// TwinCAT 3 PLC project Xplanar
// ProgramVersion: 3.1.4026.9
// CompilerDefines: VISU_USEPROPERTYINFO
// libraries:
//   CmpBitmapPool, * (System)
//   Tc2_Standard, * (Beckhoff Automation GmbH)
//   Tc2_System, * (Beckhoff Automation GmbH)
//   Tc2_Utilities, * (Beckhoff Automation GmbH)
//   Tc3_Mc3PlanarMotion, * (Beckhoff Automation GmbH)
//   Tc3_Physics, * (Beckhoff Automation GmbH)
//   Tc3_XPlanarUtility, * (Beckhoff Automation GmbH)
//   VisuDialogs, * (System)
//   VisuSymbols, 4.5.0.0 (System)
// project tree:
//   DUTs/ TurtleNames.TcDUT
//   / GlobalTextList.TcGTLO, ImagePool.TcIPO (not stored), PlcTask.TcTTO
//   GVLs/ GVL.TcGVL
//   POUs/ HMI_UpdateMoverStatus.TcPOU, MAIN.TcPOU, randnum.TcPOU, Traffic_Light.TcPOU, WinnersList.TcPOU, Winner_Display.TcPOU
// real-time tasks:
//   TASK XPlanar Task3: cycle T#250us, priority 1, ADS port 350
//   TASK MC-Task (MET): cycle T#2ms, priority 2, ADS port 351
//   TASK MC-Task (MPT): cycle T#10ms, priority 3, ADS port 352
//   TASK Job Task: cycle default, priority 4
//   TASK MC-Task (MET)_1: cycle T#2ms, priority 5, ADS port 521
//   TASK MC-Task (MPT)_1: cycle T#10ms, priority 10, ADS port 531
//   TASK PlcTask: cycle T#10ms, priority 20, ADS port 353
// I/O:
//   DEVICE Device 1 (EtherCAT), AmsNetId 172.18.137.9.2.1
//     Box 1 (EP2316-0003) [EP2316-0003 8 Ch. Dig. In, 10µs, 8Ch. Dig. Out 24V, 0,5A, Diagnostic, 10-Pole Plug Connector]
//   DEVICE Device 2 (EtherCAT), AmsNetId 172.18.137.9.3.1
//     Term 2 (APS4322-7000) [APS4322-7000 Drive]
//       Term 3 (APS4322-5000) [APS4322-5000 Feedback]
//     Term 4 (APS4322-7000) [APS4322-7000 Drive]
//       Term 5 (APS4322-5000) [APS4322-5000 Feedback]
// variable links:
//   Device 2 (EtherCAT) <-> TcCOM Objects/XPlanar/Part1/Tile1
//     Term 2 (APS4322-7000)/APS Comm Inputs/CommStatusWord <-> Data Pointer/MoverCommStatusWord
//     Term 2 (APS4322-7000)/APS Comm Inputs/Data {1..4} <-> Data Pointer/MoverCommDataIn[{0..3}]  (4 links)
//     Term 2 (APS4322-7000)/APS Comm Outputs/CommControlWord <-> Data Pointer/MoverCommControlWord
//     Term 2 (APS4322-7000)/APS Comm Outputs/Data 1 <-> Data Pointer/MoverCommDataOut
//     Term 2 (APS4322-7000)/APS Diagdata/DC Link Voltage <-> Data Pointer/DcLinkVoltage
//     Term 2 (APS4322-7000)/APS Diagdata/Power supply current <-> Data Pointer/PowerSupplyCurrent
//     Term 2 (APS4322-7000)/APS Inputs/StatusWord <-> Data Pointer/PowerUnitStatusWord
//     Term 2 (APS4322-7000)/APS Outputs/ControlWord <-> Data Pointer/PowerUnitControlWord
//     Term 2 (APS4322-7000)/APS Outputs/Current D 0X0 <-> Data Pointer/DCurrentSetPoints[0]
//     Term 2 (APS4322-7000)/APS Outputs/Current D 0X1 <-> Data Pointer/DCurrentSetPoints[1]
//     Term 2 (APS4322-7000)/APS Outputs/Current D 0X2 <-> Data Pointer/DCurrentSetPoints[2]
//     Term 2 (APS4322-7000)/APS Outputs/Current D 1X0 <-> Data Pointer/DCurrentSetPoints[6]
//     Term 2 (APS4322-7000)/APS Outputs/Current D 1X1 <-> Data Pointer/DCurrentSetPoints[7]
//     Term 2 (APS4322-7000)/APS Outputs/Current D 1X2 <-> Data Pointer/DCurrentSetPoints[8]
//     Term 2 (APS4322-7000)/APS Outputs/Current D 2X0 <-> Data Pointer/DCurrentSetPoints[12]
//     Term 2 (APS4322-7000)/APS Outputs/Current D 2X1 <-> Data Pointer/DCurrentSetPoints[13]
//     Term 2 (APS4322-7000)/APS Outputs/Current D 2X2 <-> Data Pointer/DCurrentSetPoints[14]
//     Term 2 (APS4322-7000)/APS Outputs/Current D 3X0 <-> Data Pointer/DCurrentSetPoints[18]
//     Term 2 (APS4322-7000)/APS Outputs/Current D 3X1 <-> Data Pointer/DCurrentSetPoints[19]
//     Term 2 (APS4322-7000)/APS Outputs/Current D 3X2 <-> Data Pointer/DCurrentSetPoints[20]
//     Term 2 (APS4322-7000)/APS Outputs/Current D 0Y0 <-> Data Pointer/DCurrentSetPoints[3]
//     Term 2 (APS4322-7000)/APS Outputs/Current D 0Y1 <-> Data Pointer/DCurrentSetPoints[4]
//     Term 2 (APS4322-7000)/APS Outputs/Current D 0Y2 <-> Data Pointer/DCurrentSetPoints[5]
//     Term 2 (APS4322-7000)/APS Outputs/Current D 1Y0 <-> Data Pointer/DCurrentSetPoints[9]
//     Term 2 (APS4322-7000)/APS Outputs/Current D 1Y1 <-> Data Pointer/DCurrentSetPoints[10]
//     Term 2 (APS4322-7000)/APS Outputs/Current D 1Y2 <-> Data Pointer/DCurrentSetPoints[11]
//     Term 2 (APS4322-7000)/APS Outputs/Current D 2Y0 <-> Data Pointer/DCurrentSetPoints[15]
//     Term 2 (APS4322-7000)/APS Outputs/Current D 2Y1 <-> Data Pointer/DCurrentSetPoints[16]
//     Term 2 (APS4322-7000)/APS Outputs/Current D 2Y2 <-> Data Pointer/DCurrentSetPoints[17]
//     Term 2 (APS4322-7000)/APS Outputs/Current D 3Y0 <-> Data Pointer/DCurrentSetPoints[21]
//     Term 2 (APS4322-7000)/APS Outputs/Current D 3Y1 <-> Data Pointer/DCurrentSetPoints[22]
//     Term 2 (APS4322-7000)/APS Outputs/Current D 3Y2 <-> Data Pointer/DCurrentSetPoints[23]
//     Term 2 (APS4322-7000)/APS Outputs/Current Q 0X0 <-> Data Pointer/QCurrentSetPoints[0]
//     Term 2 (APS4322-7000)/APS Outputs/Current Q 0X1 <-> Data Pointer/QCurrentSetPoints[1]
//     Term 2 (APS4322-7000)/APS Outputs/Current Q 0X2 <-> Data Pointer/QCurrentSetPoints[2]
//     Term 2 (APS4322-7000)/APS Outputs/Current Q 1X0 <-> Data Pointer/QCurrentSetPoints[6]
//     Term 2 (APS4322-7000)/APS Outputs/Current Q 1X1 <-> Data Pointer/QCurrentSetPoints[7]
//     Term 2 (APS4322-7000)/APS Outputs/Current Q 1X2 <-> Data Pointer/QCurrentSetPoints[8]
//     Term 2 (APS4322-7000)/APS Outputs/Current Q 2X0 <-> Data Pointer/QCurrentSetPoints[12]
//     Term 2 (APS4322-7000)/APS Outputs/Current Q 2X1 <-> Data Pointer/QCurrentSetPoints[13]
//     Term 2 (APS4322-7000)/APS Outputs/Current Q 2X2 <-> Data Pointer/QCurrentSetPoints[14]
//     Term 2 (APS4322-7000)/APS Outputs/Current Q 3X0 <-> Data Pointer/QCurrentSetPoints[18]
//     Term 2 (APS4322-7000)/APS Outputs/Current Q 3X1 <-> Data Pointer/QCurrentSetPoints[19]
//     Term 2 (APS4322-7000)/APS Outputs/Current Q 3X2 <-> Data Pointer/QCurrentSetPoints[20]
//     Term 2 (APS4322-7000)/APS Outputs/Current Q 0Y0 <-> Data Pointer/QCurrentSetPoints[3]
//     Term 2 (APS4322-7000)/APS Outputs/Current Q 0Y1 <-> Data Pointer/QCurrentSetPoints[4]
//     Term 2 (APS4322-7000)/APS Outputs/Current Q 0Y2 <-> Data Pointer/QCurrentSetPoints[5]
//     Term 2 (APS4322-7000)/APS Outputs/Current Q 1Y0 <-> Data Pointer/QCurrentSetPoints[9]
//     Term 2 (APS4322-7000)/APS Outputs/Current Q 1Y1 <-> Data Pointer/QCurrentSetPoints[10]
//     Term 2 (APS4322-7000)/APS Outputs/Current Q 1Y2 <-> Data Pointer/QCurrentSetPoints[11]
//     Term 2 (APS4322-7000)/APS Outputs/Current Q 2Y0 <-> Data Pointer/QCurrentSetPoints[15]
//     Term 2 (APS4322-7000)/APS Outputs/Current Q 2Y1 <-> Data Pointer/QCurrentSetPoints[16]
//     Term 2 (APS4322-7000)/APS Outputs/Current Q 2Y2 <-> Data Pointer/QCurrentSetPoints[17]
//     Term 2 (APS4322-7000)/APS Outputs/Current Q 3Y0 <-> Data Pointer/QCurrentSetPoints[21]
//     Term 2 (APS4322-7000)/APS Outputs/Current Q 3Y1 <-> Data Pointer/QCurrentSetPoints[22]
//     Term 2 (APS4322-7000)/APS Outputs/Current Q 3Y2 <-> Data Pointer/QCurrentSetPoints[23]
//     Term 2 (APS4322-7000)/APS Outputs/PhiE 0X0 <-> Data Pointer/PhiSetPoints[0]
//     Term 2 (APS4322-7000)/APS Outputs/PhiE 0X1 <-> Data Pointer/PhiSetPoints[1]
//     Term 2 (APS4322-7000)/APS Outputs/PhiE 0X2 <-> Data Pointer/PhiSetPoints[2]
//     Term 2 (APS4322-7000)/APS Outputs/PhiE 1X0 <-> Data Pointer/PhiSetPoints[6]
//     Term 2 (APS4322-7000)/APS Outputs/PhiE 1X1 <-> Data Pointer/PhiSetPoints[7]
//     Term 2 (APS4322-7000)/APS Outputs/PhiE 1X2 <-> Data Pointer/PhiSetPoints[8]
//     Term 2 (APS4322-7000)/APS Outputs/PhiE 2X0 <-> Data Pointer/PhiSetPoints[12]
//     Term 2 (APS4322-7000)/APS Outputs/PhiE 2X1 <-> Data Pointer/PhiSetPoints[13]
//     Term 2 (APS4322-7000)/APS Outputs/PhiE 2X2 <-> Data Pointer/PhiSetPoints[14]
//     Term 2 (APS4322-7000)/APS Outputs/PhiE 3X0 <-> Data Pointer/PhiSetPoints[18]
//     Term 2 (APS4322-7000)/APS Outputs/PhiE 3X1 <-> Data Pointer/PhiSetPoints[19]
//     Term 2 (APS4322-7000)/APS Outputs/PhiE 3X2 <-> Data Pointer/PhiSetPoints[20]
//     Term 2 (APS4322-7000)/APS Outputs/PhiE 0Y0 <-> Data Pointer/PhiSetPoints[3]
//     Term 2 (APS4322-7000)/APS Outputs/PhiE 0Y1 <-> Data Pointer/PhiSetPoints[4]
//     Term 2 (APS4322-7000)/APS Outputs/PhiE 0Y2 <-> Data Pointer/PhiSetPoints[5]
//     Term 2 (APS4322-7000)/APS Outputs/PhiE 1Y0 <-> Data Pointer/PhiSetPoints[9]
//     Term 2 (APS4322-7000)/APS Outputs/PhiE 1Y1 <-> Data Pointer/PhiSetPoints[10]
//     Term 2 (APS4322-7000)/APS Outputs/PhiE 1Y2 <-> Data Pointer/PhiSetPoints[11]
//     Term 2 (APS4322-7000)/APS Outputs/PhiE 2Y0 <-> Data Pointer/PhiSetPoints[15]
//     Term 2 (APS4322-7000)/APS Outputs/PhiE 2Y1 <-> Data Pointer/PhiSetPoints[16]
//     Term 2 (APS4322-7000)/APS Outputs/PhiE 2Y2 <-> Data Pointer/PhiSetPoints[17]
//     Term 2 (APS4322-7000)/APS Outputs/PhiE 3Y0 <-> Data Pointer/PhiSetPoints[21]
//     Term 2 (APS4322-7000)/APS Outputs/PhiE 3Y1 <-> Data Pointer/PhiSetPoints[22]
//     Term 2 (APS4322-7000)/APS Outputs/PhiE 3Y2 <-> Data Pointer/PhiSetPoints[23]
//     Term 2 (APS4322-7000)/Term 3 (APS4322-5000)/FB Inputs/A{0..8 step 2} X-Field <-> Data Pointer/HallSensorFieldsXYZ[{0..12 step 3}]  (5 links)
//     Term 2 (APS4322-7000)/Term 3 (APS4322-5000)/FB Inputs/A{0..8 step 2} Y-Field <-> Data Pointer/HallSensorFieldsXYZ[{1..13 step 3}]  (5 links)
//     Term 2 (APS4322-7000)/Term 3 (APS4322-5000)/FB Inputs/A{0..8 step 2} Z-Field <-> Data Pointer/HallSensorFieldsXYZ[{2..14 step 3}]  (5 links)
//     Term 2 (APS4322-7000)/Term 3 (APS4322-5000)/FB Inputs/B{1..9 step 2} X-Field <-> Data Pointer/HallSensorFieldsXYZ[{15..27 step 3}]  (5 links)
//     Term 2 (APS4322-7000)/Term 3 (APS4322-5000)/FB Inputs/B{1..9 step 2} Y-Field <-> Data Pointer/HallSensorFieldsXYZ[{16..28 step 3}]  (5 links)
//     Term 2 (APS4322-7000)/Term 3 (APS4322-5000)/FB Inputs/B{1..9 step 2} Z-Field <-> Data Pointer/HallSensorFieldsXYZ[{17..29 step 3}]  (5 links)
//     Term 2 (APS4322-7000)/Term 3 (APS4322-5000)/FB Inputs/C{0..8 step 2} X-Field <-> Data Pointer/HallSensorFieldsXYZ[{30..42 step 3}]  (5 links)
//     Term 2 (APS4322-7000)/Term 3 (APS4322-5000)/FB Inputs/C{0..8 step 2} Y-Field <-> Data Pointer/HallSensorFieldsXYZ[{31..43 step 3}]  (5 links)
//     Term 2 (APS4322-7000)/Term 3 (APS4322-5000)/FB Inputs/C{0..8 step 2} Z-Field <-> Data Pointer/HallSensorFieldsXYZ[{32..44 step 3}]  (5 links)
//     Term 2 (APS4322-7000)/Term 3 (APS4322-5000)/FB Inputs/D{1..9 step 2} X-Field <-> Data Pointer/HallSensorFieldsXYZ[{45..57 step 3}]  (5 links)
//     Term 2 (APS4322-7000)/Term 3 (APS4322-5000)/FB Inputs/D{1..9 step 2} Y-Field <-> Data Pointer/HallSensorFieldsXYZ[{46..58 step 3}]  (5 links)
//     Term 2 (APS4322-7000)/Term 3 (APS4322-5000)/FB Inputs/D{1..9 step 2} Z-Field <-> Data Pointer/HallSensorFieldsXYZ[{47..59 step 3}]  (5 links)
//     Term 2 (APS4322-7000)/Term 3 (APS4322-5000)/FB Inputs/E{0..8 step 2} X-Field <-> Data Pointer/HallSensorFieldsXYZ[{60..72 step 3}]  (5 links)
//     Term 2 (APS4322-7000)/Term 3 (APS4322-5000)/FB Inputs/E{0..8 step 2} Y-Field <-> Data Pointer/HallSensorFieldsXYZ[{61..73 step 3}]  (5 links)
//     Term 2 (APS4322-7000)/Term 3 (APS4322-5000)/FB Inputs/E{0..8 step 2} Z-Field <-> Data Pointer/HallSensorFieldsXYZ[{62..74 step 3}]  (5 links)
//     Term 2 (APS4322-7000)/Term 3 (APS4322-5000)/FB Inputs/F{1..9 step 2} X-Field <-> Data Pointer/HallSensorFieldsXYZ[{75..87 step 3}]  (5 links)
//     Term 2 (APS4322-7000)/Term 3 (APS4322-5000)/FB Inputs/F{1..9 step 2} Y-Field <-> Data Pointer/HallSensorFieldsXYZ[{76..88 step 3}]  (5 links)
//     Term 2 (APS4322-7000)/Term 3 (APS4322-5000)/FB Inputs/F{1..9 step 2} Z-Field <-> Data Pointer/HallSensorFieldsXYZ[{77..89 step 3}]  (5 links)
//     Term 2 (APS4322-7000)/Term 3 (APS4322-5000)/FB Inputs/G{0..8 step 2} X-Field <-> Data Pointer/HallSensorFieldsXYZ[{90..102 step 3}]  (5 links)
//     Term 2 (APS4322-7000)/Term 3 (APS4322-5000)/FB Inputs/G{0..8 step 2} Y-Field <-> Data Pointer/HallSensorFieldsXYZ[{91..103 step 3}]  (5 links)
//     Term 2 (APS4322-7000)/Term 3 (APS4322-5000)/FB Inputs/G{0..8 step 2} Z-Field <-> Data Pointer/HallSensorFieldsXYZ[{92..104 step 3}]  (5 links)
//     Term 2 (APS4322-7000)/Term 3 (APS4322-5000)/FB Inputs/H{1..9 step 2} X-Field <-> Data Pointer/HallSensorFieldsXYZ[{105..117 step 3}]  (5 links)
//     Term 2 (APS4322-7000)/Term 3 (APS4322-5000)/FB Inputs/H{1..9 step 2} Y-Field <-> Data Pointer/HallSensorFieldsXYZ[{106..118 step 3}]  (5 links)
//     Term 2 (APS4322-7000)/Term 3 (APS4322-5000)/FB Inputs/H{1..9 step 2} Z-Field <-> Data Pointer/HallSensorFieldsXYZ[{107..119 step 3}]  (5 links)
//     Term 2 (APS4322-7000)/Term 3 (APS4322-5000)/FB Inputs/I{0..8 step 2} X-Field <-> Data Pointer/HallSensorFieldsXYZ[{120..132 step 3}]  (5 links)
//     Term 2 (APS4322-7000)/Term 3 (APS4322-5000)/FB Inputs/I{0..8 step 2} Y-Field <-> Data Pointer/HallSensorFieldsXYZ[{121..133 step 3}]  (5 links)
//     Term 2 (APS4322-7000)/Term 3 (APS4322-5000)/FB Inputs/I{0..8 step 2} Z-Field <-> Data Pointer/HallSensorFieldsXYZ[{122..134 step 3}]  (5 links)
//     Term 2 (APS4322-7000)/Term 3 (APS4322-5000)/FB Inputs/J{1..9 step 2} X-Field <-> Data Pointer/HallSensorFieldsXYZ[{135..147 step 3}]  (5 links)
//     Term 2 (APS4322-7000)/Term 3 (APS4322-5000)/FB Inputs/J{1..9 step 2} Y-Field <-> Data Pointer/HallSensorFieldsXYZ[{136..148 step 3}]  (5 links)
//     Term 2 (APS4322-7000)/Term 3 (APS4322-5000)/FB Inputs/J{1..9 step 2} Z-Field <-> Data Pointer/HallSensorFieldsXYZ[{137..149 step 3}]  (5 links)
//     Term 2 (APS4322-7000)/Term 3 (APS4322-5000)/FB Inputs/Status <-> Data Pointer/FeedbackStatus
//   Device 2 (EtherCAT) <-> TcCOM Objects/XPlanar/Part1/Tile2
//     Term 4 (APS4322-7000)/APS Comm Inputs/CommStatusWord <-> Data Pointer/MoverCommStatusWord
//     Term 4 (APS4322-7000)/APS Comm Inputs/Data {1..4} <-> Data Pointer/MoverCommDataIn[{0..3}]  (4 links)
//     Term 4 (APS4322-7000)/APS Comm Outputs/CommControlWord <-> Data Pointer/MoverCommControlWord
//     Term 4 (APS4322-7000)/APS Comm Outputs/Data 1 <-> Data Pointer/MoverCommDataOut
//     Term 4 (APS4322-7000)/APS Diagdata/DC Link Voltage <-> Data Pointer/DcLinkVoltage
//     Term 4 (APS4322-7000)/APS Diagdata/Power supply current <-> Data Pointer/PowerSupplyCurrent
//     Term 4 (APS4322-7000)/APS Inputs/StatusWord <-> Data Pointer/PowerUnitStatusWord
//     Term 4 (APS4322-7000)/APS Outputs/ControlWord <-> Data Pointer/PowerUnitControlWord
//     Term 4 (APS4322-7000)/APS Outputs/Current D 0X0 <-> Data Pointer/DCurrentSetPoints[0]
//     Term 4 (APS4322-7000)/APS Outputs/Current D 0X1 <-> Data Pointer/DCurrentSetPoints[1]
//     Term 4 (APS4322-7000)/APS Outputs/Current D 0X2 <-> Data Pointer/DCurrentSetPoints[2]
//     Term 4 (APS4322-7000)/APS Outputs/Current D 1X0 <-> Data Pointer/DCurrentSetPoints[6]
//     Term 4 (APS4322-7000)/APS Outputs/Current D 1X1 <-> Data Pointer/DCurrentSetPoints[7]
//     Term 4 (APS4322-7000)/APS Outputs/Current D 1X2 <-> Data Pointer/DCurrentSetPoints[8]
//     Term 4 (APS4322-7000)/APS Outputs/Current D 2X0 <-> Data Pointer/DCurrentSetPoints[12]
//     Term 4 (APS4322-7000)/APS Outputs/Current D 2X1 <-> Data Pointer/DCurrentSetPoints[13]
//     Term 4 (APS4322-7000)/APS Outputs/Current D 2X2 <-> Data Pointer/DCurrentSetPoints[14]
//     Term 4 (APS4322-7000)/APS Outputs/Current D 3X0 <-> Data Pointer/DCurrentSetPoints[18]
//     Term 4 (APS4322-7000)/APS Outputs/Current D 3X1 <-> Data Pointer/DCurrentSetPoints[19]
//     Term 4 (APS4322-7000)/APS Outputs/Current D 3X2 <-> Data Pointer/DCurrentSetPoints[20]
//     Term 4 (APS4322-7000)/APS Outputs/Current D 0Y0 <-> Data Pointer/DCurrentSetPoints[3]
//     Term 4 (APS4322-7000)/APS Outputs/Current D 0Y1 <-> Data Pointer/DCurrentSetPoints[4]
//     Term 4 (APS4322-7000)/APS Outputs/Current D 0Y2 <-> Data Pointer/DCurrentSetPoints[5]
//     Term 4 (APS4322-7000)/APS Outputs/Current D 1Y0 <-> Data Pointer/DCurrentSetPoints[9]
//     Term 4 (APS4322-7000)/APS Outputs/Current D 1Y1 <-> Data Pointer/DCurrentSetPoints[10]
//     Term 4 (APS4322-7000)/APS Outputs/Current D 1Y2 <-> Data Pointer/DCurrentSetPoints[11]
//     Term 4 (APS4322-7000)/APS Outputs/Current D 2Y0 <-> Data Pointer/DCurrentSetPoints[15]
//     Term 4 (APS4322-7000)/APS Outputs/Current D 2Y1 <-> Data Pointer/DCurrentSetPoints[16]
//     Term 4 (APS4322-7000)/APS Outputs/Current D 2Y2 <-> Data Pointer/DCurrentSetPoints[17]
//     Term 4 (APS4322-7000)/APS Outputs/Current D 3Y0 <-> Data Pointer/DCurrentSetPoints[21]
//     Term 4 (APS4322-7000)/APS Outputs/Current D 3Y1 <-> Data Pointer/DCurrentSetPoints[22]
//     Term 4 (APS4322-7000)/APS Outputs/Current D 3Y2 <-> Data Pointer/DCurrentSetPoints[23]
//     Term 4 (APS4322-7000)/APS Outputs/Current Q 0X0 <-> Data Pointer/QCurrentSetPoints[0]
//     Term 4 (APS4322-7000)/APS Outputs/Current Q 0X1 <-> Data Pointer/QCurrentSetPoints[1]
//     Term 4 (APS4322-7000)/APS Outputs/Current Q 0X2 <-> Data Pointer/QCurrentSetPoints[2]
//     Term 4 (APS4322-7000)/APS Outputs/Current Q 1X0 <-> Data Pointer/QCurrentSetPoints[6]
//     Term 4 (APS4322-7000)/APS Outputs/Current Q 1X1 <-> Data Pointer/QCurrentSetPoints[7]
//     Term 4 (APS4322-7000)/APS Outputs/Current Q 1X2 <-> Data Pointer/QCurrentSetPoints[8]
//     Term 4 (APS4322-7000)/APS Outputs/Current Q 2X0 <-> Data Pointer/QCurrentSetPoints[12]
//     Term 4 (APS4322-7000)/APS Outputs/Current Q 2X1 <-> Data Pointer/QCurrentSetPoints[13]
//     Term 4 (APS4322-7000)/APS Outputs/Current Q 2X2 <-> Data Pointer/QCurrentSetPoints[14]
//     Term 4 (APS4322-7000)/APS Outputs/Current Q 3X0 <-> Data Pointer/QCurrentSetPoints[18]
//     Term 4 (APS4322-7000)/APS Outputs/Current Q 3X1 <-> Data Pointer/QCurrentSetPoints[19]
//     Term 4 (APS4322-7000)/APS Outputs/Current Q 3X2 <-> Data Pointer/QCurrentSetPoints[20]
//     Term 4 (APS4322-7000)/APS Outputs/Current Q 0Y0 <-> Data Pointer/QCurrentSetPoints[3]
//     Term 4 (APS4322-7000)/APS Outputs/Current Q 0Y1 <-> Data Pointer/QCurrentSetPoints[4]
//     Term 4 (APS4322-7000)/APS Outputs/Current Q 0Y2 <-> Data Pointer/QCurrentSetPoints[5]
//     Term 4 (APS4322-7000)/APS Outputs/Current Q 1Y0 <-> Data Pointer/QCurrentSetPoints[9]
//     Term 4 (APS4322-7000)/APS Outputs/Current Q 1Y1 <-> Data Pointer/QCurrentSetPoints[10]
//     Term 4 (APS4322-7000)/APS Outputs/Current Q 1Y2 <-> Data Pointer/QCurrentSetPoints[11]
//     Term 4 (APS4322-7000)/APS Outputs/Current Q 2Y0 <-> Data Pointer/QCurrentSetPoints[15]
//     Term 4 (APS4322-7000)/APS Outputs/Current Q 2Y1 <-> Data Pointer/QCurrentSetPoints[16]
//     Term 4 (APS4322-7000)/APS Outputs/Current Q 2Y2 <-> Data Pointer/QCurrentSetPoints[17]
//     Term 4 (APS4322-7000)/APS Outputs/Current Q 3Y0 <-> Data Pointer/QCurrentSetPoints[21]
//     Term 4 (APS4322-7000)/APS Outputs/Current Q 3Y1 <-> Data Pointer/QCurrentSetPoints[22]
//     Term 4 (APS4322-7000)/APS Outputs/Current Q 3Y2 <-> Data Pointer/QCurrentSetPoints[23]
//     Term 4 (APS4322-7000)/APS Outputs/PhiE 0X0 <-> Data Pointer/PhiSetPoints[0]
//     Term 4 (APS4322-7000)/APS Outputs/PhiE 0X1 <-> Data Pointer/PhiSetPoints[1]
//     Term 4 (APS4322-7000)/APS Outputs/PhiE 0X2 <-> Data Pointer/PhiSetPoints[2]
//     Term 4 (APS4322-7000)/APS Outputs/PhiE 1X0 <-> Data Pointer/PhiSetPoints[6]
//     Term 4 (APS4322-7000)/APS Outputs/PhiE 1X1 <-> Data Pointer/PhiSetPoints[7]
//     Term 4 (APS4322-7000)/APS Outputs/PhiE 1X2 <-> Data Pointer/PhiSetPoints[8]
//     Term 4 (APS4322-7000)/APS Outputs/PhiE 2X0 <-> Data Pointer/PhiSetPoints[12]
//     Term 4 (APS4322-7000)/APS Outputs/PhiE 2X1 <-> Data Pointer/PhiSetPoints[13]
//     Term 4 (APS4322-7000)/APS Outputs/PhiE 2X2 <-> Data Pointer/PhiSetPoints[14]
//     Term 4 (APS4322-7000)/APS Outputs/PhiE 3X0 <-> Data Pointer/PhiSetPoints[18]
//     Term 4 (APS4322-7000)/APS Outputs/PhiE 3X1 <-> Data Pointer/PhiSetPoints[19]
//     Term 4 (APS4322-7000)/APS Outputs/PhiE 3X2 <-> Data Pointer/PhiSetPoints[20]
//     Term 4 (APS4322-7000)/APS Outputs/PhiE 0Y0 <-> Data Pointer/PhiSetPoints[3]
//     Term 4 (APS4322-7000)/APS Outputs/PhiE 0Y1 <-> Data Pointer/PhiSetPoints[4]
//     Term 4 (APS4322-7000)/APS Outputs/PhiE 0Y2 <-> Data Pointer/PhiSetPoints[5]
//     Term 4 (APS4322-7000)/APS Outputs/PhiE 1Y0 <-> Data Pointer/PhiSetPoints[9]
//     Term 4 (APS4322-7000)/APS Outputs/PhiE 1Y1 <-> Data Pointer/PhiSetPoints[10]
//     Term 4 (APS4322-7000)/APS Outputs/PhiE 1Y2 <-> Data Pointer/PhiSetPoints[11]
//     Term 4 (APS4322-7000)/APS Outputs/PhiE 2Y0 <-> Data Pointer/PhiSetPoints[15]
//     Term 4 (APS4322-7000)/APS Outputs/PhiE 2Y1 <-> Data Pointer/PhiSetPoints[16]
//     Term 4 (APS4322-7000)/APS Outputs/PhiE 2Y2 <-> Data Pointer/PhiSetPoints[17]
//     Term 4 (APS4322-7000)/APS Outputs/PhiE 3Y0 <-> Data Pointer/PhiSetPoints[21]
//     Term 4 (APS4322-7000)/APS Outputs/PhiE 3Y1 <-> Data Pointer/PhiSetPoints[22]
//     Term 4 (APS4322-7000)/APS Outputs/PhiE 3Y2 <-> Data Pointer/PhiSetPoints[23]
//     Term 4 (APS4322-7000)/Term 5 (APS4322-5000)/FB Inputs/A{0..8 step 2} X-Field <-> Data Pointer/HallSensorFieldsXYZ[{0..12 step 3}]  (5 links)
//     Term 4 (APS4322-7000)/Term 5 (APS4322-5000)/FB Inputs/A{0..8 step 2} Y-Field <-> Data Pointer/HallSensorFieldsXYZ[{1..13 step 3}]  (5 links)
//     Term 4 (APS4322-7000)/Term 5 (APS4322-5000)/FB Inputs/A{0..8 step 2} Z-Field <-> Data Pointer/HallSensorFieldsXYZ[{2..14 step 3}]  (5 links)
//     Term 4 (APS4322-7000)/Term 5 (APS4322-5000)/FB Inputs/B{1..9 step 2} X-Field <-> Data Pointer/HallSensorFieldsXYZ[{15..27 step 3}]  (5 links)
//     Term 4 (APS4322-7000)/Term 5 (APS4322-5000)/FB Inputs/B{1..9 step 2} Y-Field <-> Data Pointer/HallSensorFieldsXYZ[{16..28 step 3}]  (5 links)
//     Term 4 (APS4322-7000)/Term 5 (APS4322-5000)/FB Inputs/B{1..9 step 2} Z-Field <-> Data Pointer/HallSensorFieldsXYZ[{17..29 step 3}]  (5 links)
//     Term 4 (APS4322-7000)/Term 5 (APS4322-5000)/FB Inputs/C{0..8 step 2} X-Field <-> Data Pointer/HallSensorFieldsXYZ[{30..42 step 3}]  (5 links)
//     Term 4 (APS4322-7000)/Term 5 (APS4322-5000)/FB Inputs/C{0..8 step 2} Y-Field <-> Data Pointer/HallSensorFieldsXYZ[{31..43 step 3}]  (5 links)
//     Term 4 (APS4322-7000)/Term 5 (APS4322-5000)/FB Inputs/C{0..8 step 2} Z-Field <-> Data Pointer/HallSensorFieldsXYZ[{32..44 step 3}]  (5 links)
//     Term 4 (APS4322-7000)/Term 5 (APS4322-5000)/FB Inputs/D{1..9 step 2} X-Field <-> Data Pointer/HallSensorFieldsXYZ[{45..57 step 3}]  (5 links)
//     Term 4 (APS4322-7000)/Term 5 (APS4322-5000)/FB Inputs/D{1..9 step 2} Y-Field <-> Data Pointer/HallSensorFieldsXYZ[{46..58 step 3}]  (5 links)
//     Term 4 (APS4322-7000)/Term 5 (APS4322-5000)/FB Inputs/D{1..9 step 2} Z-Field <-> Data Pointer/HallSensorFieldsXYZ[{47..59 step 3}]  (5 links)
//     Term 4 (APS4322-7000)/Term 5 (APS4322-5000)/FB Inputs/E{0..8 step 2} X-Field <-> Data Pointer/HallSensorFieldsXYZ[{60..72 step 3}]  (5 links)
//     Term 4 (APS4322-7000)/Term 5 (APS4322-5000)/FB Inputs/E{0..8 step 2} Y-Field <-> Data Pointer/HallSensorFieldsXYZ[{61..73 step 3}]  (5 links)
//     Term 4 (APS4322-7000)/Term 5 (APS4322-5000)/FB Inputs/E{0..8 step 2} Z-Field <-> Data Pointer/HallSensorFieldsXYZ[{62..74 step 3}]  (5 links)
//     Term 4 (APS4322-7000)/Term 5 (APS4322-5000)/FB Inputs/F{1..9 step 2} X-Field <-> Data Pointer/HallSensorFieldsXYZ[{75..87 step 3}]  (5 links)
//     Term 4 (APS4322-7000)/Term 5 (APS4322-5000)/FB Inputs/F{1..9 step 2} Y-Field <-> Data Pointer/HallSensorFieldsXYZ[{76..88 step 3}]  (5 links)
//     Term 4 (APS4322-7000)/Term 5 (APS4322-5000)/FB Inputs/F{1..9 step 2} Z-Field <-> Data Pointer/HallSensorFieldsXYZ[{77..89 step 3}]  (5 links)
//     Term 4 (APS4322-7000)/Term 5 (APS4322-5000)/FB Inputs/G{0..8 step 2} X-Field <-> Data Pointer/HallSensorFieldsXYZ[{90..102 step 3}]  (5 links)
//     Term 4 (APS4322-7000)/Term 5 (APS4322-5000)/FB Inputs/G{0..8 step 2} Y-Field <-> Data Pointer/HallSensorFieldsXYZ[{91..103 step 3}]  (5 links)
//     Term 4 (APS4322-7000)/Term 5 (APS4322-5000)/FB Inputs/G{0..8 step 2} Z-Field <-> Data Pointer/HallSensorFieldsXYZ[{92..104 step 3}]  (5 links)
//     Term 4 (APS4322-7000)/Term 5 (APS4322-5000)/FB Inputs/H{1..9 step 2} X-Field <-> Data Pointer/HallSensorFieldsXYZ[{105..117 step 3}]  (5 links)
//     Term 4 (APS4322-7000)/Term 5 (APS4322-5000)/FB Inputs/H{1..9 step 2} Y-Field <-> Data Pointer/HallSensorFieldsXYZ[{106..118 step 3}]  (5 links)
//     Term 4 (APS4322-7000)/Term 5 (APS4322-5000)/FB Inputs/H{1..9 step 2} Z-Field <-> Data Pointer/HallSensorFieldsXYZ[{107..119 step 3}]  (5 links)
//     Term 4 (APS4322-7000)/Term 5 (APS4322-5000)/FB Inputs/I{0..8 step 2} X-Field <-> Data Pointer/HallSensorFieldsXYZ[{120..132 step 3}]  (5 links)
//     Term 4 (APS4322-7000)/Term 5 (APS4322-5000)/FB Inputs/I{0..8 step 2} Y-Field <-> Data Pointer/HallSensorFieldsXYZ[{121..133 step 3}]  (5 links)
//     Term 4 (APS4322-7000)/Term 5 (APS4322-5000)/FB Inputs/I{0..8 step 2} Z-Field <-> Data Pointer/HallSensorFieldsXYZ[{122..134 step 3}]  (5 links)
//     Term 4 (APS4322-7000)/Term 5 (APS4322-5000)/FB Inputs/J{1..9 step 2} X-Field <-> Data Pointer/HallSensorFieldsXYZ[{135..147 step 3}]  (5 links)
//     Term 4 (APS4322-7000)/Term 5 (APS4322-5000)/FB Inputs/J{1..9 step 2} Y-Field <-> Data Pointer/HallSensorFieldsXYZ[{136..148 step 3}]  (5 links)
//     Term 4 (APS4322-7000)/Term 5 (APS4322-5000)/FB Inputs/J{1..9 step 2} Z-Field <-> Data Pointer/HallSensorFieldsXYZ[{137..149 step 3}]  (5 links)
//     Term 4 (APS4322-7000)/Term 5 (APS4322-5000)/FB Inputs/Status <-> Data Pointer/FeedbackStatus
//   XPlanar MC Project/Axes/Mover4220_1 <-> TcCOM Objects/XPlanar/Mover4220_1
//     IoToMc/STD <-> OutputsToNC3/HWToNC3
//     McToIo/STD <-> InputsFromNC3/NC3ToHW
//   XPlanar MC Project/Axes/Mover4220_2 <-> TcCOM Objects/XPlanar/Mover4220_2
//     IoToMc/STD <-> OutputsToNC3/HWToNC3
//     McToIo/STD <-> InputsFromNC3/NC3ToHW
//   Xplanar/Xplanar Instance <-> XPlanar MC Project/Axes/Mover4220_1
//     PlcTask Inputs/GVL.fbMover.MCTOPLC/ACT <-> McToPlc/ACT
//     PlcTask Inputs/GVL.fbMover.MCTOPLC/COORDMODE <-> McToPlc/COORDMODE
//     PlcTask Inputs/GVL.fbMover.MCTOPLC/SET <-> McToPlc/SET
//     PlcTask Inputs/GVL.fbMover.MCTOPLC/SETONTRACK <-> McToPlc/SETONTRACK
//     PlcTask Inputs/GVL.fbMover.MCTOPLC/STD <-> McToPlc/STD
//     PlcTask Outputs/GVL.fbMover.PLCTOMC/STD <-> PlcToMc/STD
//   Xplanar/Xplanar Instance <-> XPlanar MC Project/Axes/Mover4220_2
//     PlcTask Inputs/GVL.fbMover2.MCTOPLC/ACT <-> McToPlc/ACT
//     PlcTask Inputs/GVL.fbMover2.MCTOPLC/COORDMODE <-> McToPlc/COORDMODE
//     PlcTask Inputs/GVL.fbMover2.MCTOPLC/SET <-> McToPlc/SET
//     PlcTask Inputs/GVL.fbMover2.MCTOPLC/SETONTRACK <-> McToPlc/SETONTRACK
//     PlcTask Inputs/GVL.fbMover2.MCTOPLC/STD <-> McToPlc/STD
//     PlcTask Outputs/GVL.fbMover2.PLCTOMC/STD <-> PlcToMc/STD

CONFIGURATION Xplanar
    RESOURCE PLC ON TwinCAT3
        TASK PlcTask(INTERVAL := T#10ms, PRIORITY := 20);
        PROGRAM MAIN WITH PlcTask : MAIN;
    END_RESOURCE
END_CONFIGURATION

// ---- DUTs/TurtleNames.TcDUT
{attribute 'qualified_only'}
{attribute 'strict'}
{attribute 'to_string'}
TYPE TurtleNames :
(
	Batman := 1,Superman:=2
);
END_TYPE

// ---- GVLs/GVL.TcGVL
//{attribute 'qualified_only'}
VAR_GLOBAL
	bEnable: BOOL;
	BEGIN : BOOL;
	bDisable: BOOL;
	bReset : BOOL;
	Ready : BOOL;
	START_RACE: BOOL;
	nCase : UINT :=10;
	fbMover : MC_PlanarMover;
	fbMover2 : MC_PlanarMover;
	cmdFB: MC_Planarfeedback;
	cmdFB2:MC_Planarfeedback;
	cmdFB3:MC_Planarfeedback;
	cmdFB4:MC_Planarfeedback;
	stMoverState: MC_Planar_State;
	stMoverState2: MC_Planar_State;
	stMoverPositions : ARRAY [1..14] OF PositionXYC;
	fbDynMove : DynamicConstraint_PathXY;
	fbDynMoveRace1 : DynamicConstraint_PathXY;
	fbDynMoveRace2 : DynamicConstraint_PathXY;
	fbDynRotate : DynamicConstraint_Coordinates;
	stMoveCOptions : ST_MoveCOptions;
	
	randnumFB : randnum;
	RandSpeed: LREAL;
	RandSpeed2: LREAL;
	TON_Timer : TON; // Declare a TON timer instance
	TimerInterval : TIME := T#2s; // Timer interval of 1 second
	DebugLog : STRING;
	Turns : ST_MoveCOptions;
	RaceFinished : TON;
	
	
	Turtle_1_Winner : BOOL ;
	Turtle_2_Winner: BOOL;
	
	HMI_Settings_Hide : BOOL;
	
	Enabled_State: BOOL;
	Start_Button_Pressed: BOOL;
	
	Traffic_timer : tof;
	
	TlRedVisibility : STRING := 'Visible';
	TlGreenVisibility : STRING := 'Collapsed';
	TlYellowVisibility : STRING := 'Collapsed';
	
	Trigger2 : F_TRIG;
	HMI_Turtle_1_Display: STRING := 'collapsed';
	HMI_Turtle_2_Display: STRING := 'Collapsed';
END_VAR

// ---- POUs/MAIN.TcPOU
PROGRAM MAIN
VAR
	(*bEnable: BOOL;
	BEGIN : BOOL;
	bDisable: BOOL;
	bReset : BOOL;
	Ready : BOOL;
	START_RACE: BOOL;
	nCase : UINT :=10;
	fbMover : MC_PlanarMover;
	fbMover2 : MC_PlanarMover;
	cmdFB: MC_Planarfeedback;
	cmdFB2:MC_Planarfeedback;
	cmdFB3:MC_Planarfeedback;
	cmdFB4:MC_Planarfeedback;
	stMoverState: MC_Planar_State;
	stMoverState2: MC_Planar_State;
	stMoverPositions : ARRAY [1..14] OF PositionXYC;
	fbDynMove : DynamicConstraint_PathXY;
	fbDynMoveRace1 : DynamicConstraint_PathXY;
	fbDynMoveRace2 : DynamicConstraint_PathXY;
	fbDynRotate : DynamicConstraint_Coordinates;
	stMoveCOptions : ST_MoveCOptions;
	
	randnumFB : randnum;
	RandSpeed: LREAL;
	RandSpeed2: LREAL;
	TON_Timer : TON; // Declare a TON timer instance
	TimerInterval : TIME := T#2s; // Timer interval of 1 second
	DebugLog : STRING;
	Turns : ST_MoveCOptions;
	RaceFinished : TON;
	
	
	Turtle_1_Winner : BOOL ;
	Turtle_2_Winner: BOOL;
	
	HMI_Settings_Hide : BOOL;
	
	Enabled_State: BOOL;
	Start_Button_Pressed: BOOL;
	
	Traffic_timer : ton;
	
	TlRedVisibility : STRING := 'Visible';
	TlGreenVisibility : STRING := 'Collapsed';
	TlYellowVisibility : STRING := 'Collapsed';
	
	Trigger2 : F_TRIG;
	HMI_Turtle_1_Display: STRING := 'collapsed';
	HMI_Turtle_2_Display: STRING := 'Collapsed';
	*)
END_VAR

fbMover.Update();
fbMover2.Update();
cmdfb.Update();
cmdfb2.Update();
stMoverState := fbMover.MCTOPLC.STD.State;
stMoverState2 := fbMover2.MCTOPLC.STD.State;




IF bEnable THEN
	fbMover.Enable(cmdfb);
	fbMover2.Enable(cmdfb2);
	bEnable:= FALSE;
	Enabled_State := TRUE;
	
END_IF

IF bReset THEN
	fbMover.Reset(cmdFB);
	fbMover2.Reset(cmdFB2);
	breset := FALSE;
END_IF

CASE nCase OF
		
	

	10: // Initialize Race
		
		randnumFB();
		RandSpeed := randnumFB.RandomNumber;
		randnumFB();
		RandSpeed2 := randnumFB.RandomNumber;

		stMoverPositions[1].SetValuesXYC(180,70,0);
		stMoverPositions[2].SetValuesXYC(180,400,0);
		stMoverPositions[3].SetValuesXYC(176,371,0);
		
		stMoverPositions[4].SetValuesXYC(60,400,0); // top
		stMoverPositions[5].SetValuesXYC(60,70,0); // bottom
		stMoverPositions[6].SetValuesXYC(180,400,0);
		
		stMoverPositions[10].SetValuesXYC(60,200,0); //half1
		stMoverPositions[9].SetValuesXYC(180,200,0); //half2
		stMoverPositions[8].SetValuesXYC(60,400,0); //finish 1
		stMoverPositions[7].SetValuesXYC(180,400,0); //finish 2
		
		stMoverPositions[11].SetValuesXYC(120,120,0); //mid2mover 
		stMoverPositions[12].SetValuesXYC(120,360,0); //mid1mover
		stMoverPositions[13].SetValuesXYC(180,120,0); //Mover 1 Middle Offset
		stMoverPositions[14].SetValuesXYC(60,360,0); //Mover 2 Middle Offset
		
		fbDynMove.SetValuesVADJ(3000,5000,5000,50000);
		
		Turtle_1_Winner := FALSE;
		Turtle_2_Winner := FALSE;
		
		nCase:= 20;
		
	20: // Move to opposite ends for start
			fbMover.MoveZ(cmdFB3,3,fbdynmove);
			fbMover2.MoveZ(cmdFB4,3,fbdynmove);
			fbMover.Movetoposition(cmdFB,stMoverPositions[1],fbdynmove,0);
			fbMover2.Movetoposition(cmdFB2,stMoverPositions[4],fbdynmove,0);
			
			nCase := 30;
		
	30: // wait for move
		IF cmdFB.Done AND cmdFB2.Done  THEN
			nCase:=40;
		END_IF
	40: // move to start
		fbMover.Movetoposition(cmdFB,stMoverPositions[1],fbdynmove,0);
		fbMover2.Movetoposition(cmdFB2,stMoverPositions[5],fbdynmove,0);
		nCase := 50;
		
	50: // wait for move
		IF cmdFB2.Done THEN
			nCase := 60;
		END_IF
	
	60: // Start Race
		
		
		IF Start_Button_Pressed THEN
			
			randnumFB();
			RandSpeed := randnumFB.RandomNumber;
			randnumFB();
			RandSpeed2 := randnumFB.RandomNumber;
			fbDynMoveRace1.SetValuesVADJ(RandSpeed,5000,5000,25000);
			fbDynMoveRace2.SetValuesVADJ(RandSpeed2,5000,5000,25000);
			fbMover.Movetoposition(cmdFB,stMoverPositions[2],fbDynMoveRace1,0);
			fbMover2.Movetoposition(cmdFB2,stMoverPositions[4],fbDynMoveRace2,0);
			nCase := 61;
		END_IF
	61: // Variable Speed
			
	
	
			TON_Timer(IN := TRUE, PT := TimerInterval);
			IF TON_Timer.Q THEN
				randnumFB();
				RandSpeed := randnumFB.RandomNumber;
				randnumFB();
				RandSpeed2 := randnumFB.RandomNumber;
				fbDynMoveRace1.SetValuesVADJ(RandSpeed,5000,5000,25000);
				fbDynMoveRace2.SetValuesVADJ(RandSpeed2,5000,5000,25000);				
				fbMover.Movetoposition(cmdFB,stMoverPositions[2],fbdynMoverace1,0);
				fbMover2.Movetoposition(cmdFB2,stMoverPositions[4],fbDynMoveRace2,0);		
								
			
				
				
				//fbMover.Reset(cmdFB);
				//fbMover2.Reset(cmdFB2);
				TON_Timer(IN := FALSE);
				nCase := 61;
			END_IF
			
		IF 	(cmdFB.Done) AND (NOT cmdFB2.done) THEN
			Turtle_1_Winner := TRUE;
		END_IF
		IF (NOT cmdFB.done) AND (cmdFB2.Done) THEN
			Turtle_2_Winner := TRUE;
		END_IF
			
			
		IF cmdFB.Done AND cmdFB2.Done THEN
			RaceFinished(IN:= TRUE, PT:= T#2S, Q=> , ET=> );
			//START_RACE := FALSE;
			IF RaceFinished.Q THEN
				nCase := 70;
				RaceFinished.IN := FALSE;
			END_IF
		END_IF
	70: // Move to Spin OFfsets
		fbDynMove.SetValuesVADJ(1000,2000,2000,50000);
		fbMover.Movetoposition(cmdFB,stMoverPositions[13],fbdynmove,0);
		fbMover2.Movetoposition(cmdFB2,stMoverPositions[14],fbdynmove,0);
		nCase:=71;
		
	71: // Wait for Spin Offsets
		IF cmdFB.Done AND cmdFB2.Done THEN
				nCase:=72;
		END_IF
	
	72: // Move to Spin Positions
		fbMover.Movetoposition(cmdFB,stMoverPositions[11],fbdynmove,0);
		fbMover2.Movetoposition(cmdFB2,stMoverPositions[12],fbdynmove,0);
		nCase:=73;
		
	73: // Wait for Spin Positions
		IF cmdFB.Done AND cmdFB2.Done THEN
				nCase:=74;
		END_IF
		
	74: // Spin
			Turns.additionalTurns := 3;
			Turns.direction := 1;
			fbMover.MoveC(cmdFB, 360, fbdynmove, Turns);
			fbMover2.MoveC(cmdFB2, 360, fbdynmove, Turns);
			nCase:=75;
		
	75: // Wait for Spin
		IF cmdFB.Done AND cmdFB2.Done THEN
				nCase:=10;
			END_IF
	
				
END_CASE

Traffic_Light();
Winner_Display();
WinnersList();
HMI_UpdateMoverStatus();

END_PROGRAM

// ---- POUs/Traffic_Light.TcPOU
PROGRAM Traffic_Light
VAR
END_VAR

Traffic_timer.IN := Start_Button_Pressed;
Traffic_Timer.PT := T#3S;
Traffic_timer();


IF Start_Button_Pressed THEN				//Turns HMI Traffic Light Green
	TlGreenVisibility := 'visible';
	TlYellowVisibility := 'Collapsed';
	TlRedVisibility := 'Collapsed';
END_IF

IF Traffic_Timer.ET > T#0S THEN				//Turns HMI Traffic Light Yellow
	TlGreenVisibility := 'Collapsed';
	TlYellowVisibility := 'visible';
	TlRedVisibility := 'Collapsed';
END_IF

IF NOT Traffic_Timer.Q THEN					//Turns HMI Traffic Light Red
	TlGreenVisibility := 'Collapsed';
	TlYellowVisibility := 'Collapsed';
	TlRedVisibility := 'visible';
	
	Traffic_Timer.IN := FALSE;
END_IF

END_PROGRAM

// ---- POUs/Winner_Display.TcPOU
PROGRAM Winner_Display
VAR
END_VAR

IF Turtle_1_Winner THEN					//Calls HMI to display Turtle WInner Animation
	HMI_Turtle_1_Display := 'Visible';
ELSIF Turtle_2_Winner THEN
	HMI_Turtle_2_Display := 'Visible';
ELSE
	HMI_Turtle_1_Display := 'Collapsed';
	HMI_Turtle_2_Display := 'Collapsed';
END_IF

END_PROGRAM

// ---- POUs/WinnersList.TcPOU
PROGRAM WinnersList
VAR
	Trigger1 : R_Trig;
	
	Winner_Array : ARRAY [1..10] OF STRING;
	
	i: INT := 1; // WInner Array indexing number
	
END_VAR

Trigger1(CLK:= Turtle_1_Winner OR Turtle_2_Winner, Q=> );

IF Trigger1.Q THEN
	IF WInner_Array[1] <> '' THEN
		FOR i := 10 TO 2 BY -1 DO
  		Winner_Array[i] := Winner_Array[i-1];
		END_FOR 
	END_IF
	
	IF Turtle_1_Winner THEN
		Winner_Array[1] := 'Batman';
	END_IF
	IF Turtle_2_Winner THEN
		Winner_Array[1] := 'Superman';
	END_IF
END_IF

END_PROGRAM

// ---- POUs/HMI_UpdateMoverStatus.TcPOU
PROGRAM HMI_UpdateMoverStatus
VAR
	Status_Enabled : String := 'Enabled';
	Status_Disabled : STRING := '#FFFF0000';
	Status_Running : STRING := '#FF15FF00';
	Status_Error : STRING := '#FFF1FF00';
	
	Mover1State : STRING;
	Mover2State : STRING;
	
END_VAR



CASE StMoverState OF
	0://Invalid
		Mover1State := Status_Error;
	1://Disabled
		Mover1State := Status_Disabled;
	2://Enabling
Mover1State := Status_Enabled;
	3://Enabled
		Mover1State := Status_Enabled;
	4://Disabling
		Mover1State := Status_Disabled;
	5://Error
		Mover1State := Status_Error;
	6://ErrorPending
		Mover1State := Status_Error;
	7://Resetting
		Mover1State := Status_Error;
END_CASE

END_PROGRAM

// ---- POUs/randnum.TcPOU
FUNCTION_BLOCK randnum
VAR_OUTPUT
    RandomNumber : LREAL; (* Generated random number *)
END_VAR

VAR
    DRANDFB : DRAND; (* Function Block instance for generating random numbers *)
	MinValue : LREAL := 20.0; (* Minimum value of the range *)
    MaxValue : LREAL := 30.0; (* Maximum value of the range *)
END_VAR

(* Generate a random number and scale it to the desired range *)
DRANDFB(Seed := 1); (* Call to generate a random number *)
RandomNumber := MinValue + (MaxValue - MinValue) * DRANDFB.Num;

END_FUNCTION_BLOCK

// ---- GlobalTextList.TcGTLO
TEXTLIST GlobalTextList
  36 = '%s'
  523 = 'Enable'
  777 = 'Error Reset'
  977 = 'Exit'
  479 = 'Go'
  820 = 'MAIN.stMoverState'
  9 = 'Mover 1'
  964 = 'Mover 2'
  829 = 'Previous Winners'
  529 = 'Start Race'
END_TEXTLIST
